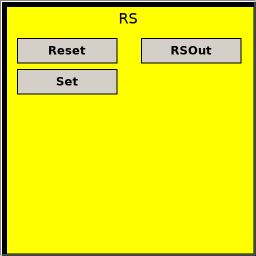
VISUALIZATION V_PH_RS  // 256x256
VAR_INPUT
	
	stSafetyRS				:ST_SAFETY_FBRS;
END_VAR
    Rectangle (2,2 256x256), colour toggle: stSafetyRS.bGeneralError
    Label (5,6 246x25), "RS"
    RoundedRectangle (17,38 100x25), "Reset", colour toggle: stSafetyRS.uStatus.stStatusWords.wInputs.8
    RoundedRectangle (141,38 100x25), "RSOut", colour toggle: stSafetyRS.uStatus.stStatusWords.wOutputs.1
    RoundedRectangle (17,69 100x25), "Set", colour toggle: stSafetyRS.uStatus.stStatusWords.wInputs.9
    Textfield (17,226 234x25), text list: 'TL_FbStateSetReset', text index: stSafetyRS.eState
END_VISUALIZATION

(* stored: Version 1.1.0.1, ProductVersion 3.1.4024.4
   Visu V_PH_RS: Id {1cf3d096-b54c-4cae-921f-8c86241afb76} *)
